PROGRAM Blinker
VAR
	
	fbBlinker1								:FB_Blinker;
	tTurnOffDelayB1							:TIME := T#1S;
	fbBlinker2								:FB_Blinker;
	
END_VAR
(* End *)

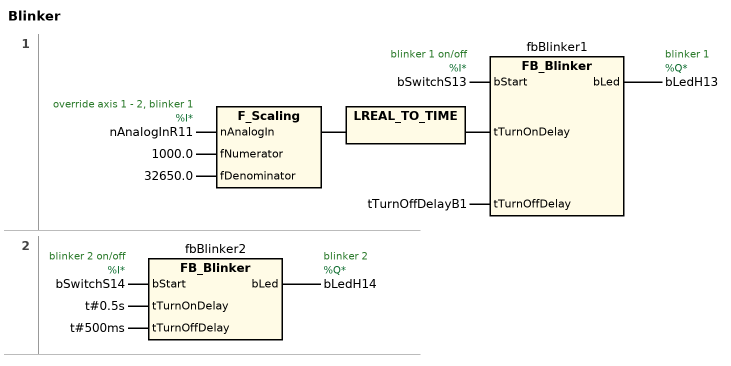
// NETWORK 1
//   bSwitchS13: blinker 1 on/off | AT %I*
//   nAnalogInR11: override axis 1 - 2, blinker 1 | AT %I*
//   bLedH13: blinker 1 | AT %Q*
fbBlinker1(
    bStart := bSwitchS13,
    tTurnOnDelay := LREAL_TO_TIME(F_Scaling(nAnalogIn := nAnalogInR11, fNumerator := 1000.0, fDenominator := 32650.0)),
    tTurnOffDelay := tTurnOffDelayB1); // FB_Blinker
bLedH13 := fbBlinker1.bLed;

// NETWORK 2
//   bSwitchS14: blinker 2 on/off | AT %I*
//   bLedH14: blinker 2 | AT %Q*
fbBlinker2(bStart := bSwitchS14, tTurnOnDelay := t#0.5s, tTurnOffDelay := t#500ms); // FB_Blinker
bLedH14 := fbBlinker2.bLed;

END_PROGRAM

(* stored: Version 1.1.0.1, ProductVersion 3.1.4022.10
   POU Blinker: Id {412a77ed-f576-470f-97fb-b89f207e2796}, SpecialFunc None *)
